{attribute 'linkalways'} 
{attribute 'no_explicit_call' := 'This FB is a CLASS and must be accessed using methods or properties'}
{attribute 'enable_dynamic_creation'}
FUNCTION_BLOCK FINAL EQ_REAL EXTENDS Node
VAR
	in1 : _REAL(0.0);
	in2 : _REAL(0.0);
	out : _BOOL(FALSE);
END_VAR

METHOD PUBLIC Clone : I_Node
VAR
	pNode : POINTER TO EQ_REAL;
END_VAR
pNode := __NEW(EQ_REAL);
Clone := pNode^;
END_METHOD

METHOD FB_init : BOOL
VAR_INPUT
	bInitRetains : BOOL; // if TRUE, the retain variables are initialized (warm start / cold start)
	bInCopyCode : BOOL;  // if TRUE, the instance afterwards gets moved into the copy code (online change)
END_VAR
AddInput('in1',THIS^.in1);
AddInput('in2',THIS^.in2);
AddOutput('out', THIS^.out);
END_METHOD

METHOD PROTECTED OnExecute
VAR
END_VAR
out.Value := in1.Value = in2.Value;
END_METHOD

END_FUNCTION_BLOCK

(* stored: Version 1.1.0.1, ProductVersion 3.1.4024.15
   POU EQ_REAL: Id {52099f19-6f47-4011-9dd5-b015d9b76a44}, SpecialFunc None
   Folder Constructor: Id {0d1e1c1c-391a-4944-8703-5215d7e66ad6}
   Method Clone: Id {cd0fc6f3-8689-40e2-903d-8b3e8f38fbc5}
   Method FB_init: Id {8a9ecbe8-45d6-4784-a968-82d36e553aff}
   Method OnExecute: Id {fb9cd043-709c-41da-8273-e18d1483862a} *)
